FUNCTION_BLOCK FIELDBUS_INT_TO_SIGNAL (* Mirrors IN->OUT if Signal Valid. *)
  (* Standard: 61499-1 *)
  (* Version 1.0, 2026-05-31, franz *)
  PACKAGE logiBUS::signalprocessing::fieldbus;
  IMPORT signalprocessing::FIELDBUS_SIGNAL::NOT_AVAILABLE_WM;
  IMPORT signalprocessing::FIELDBUS_SIGNAL::VALID_SIGNAL_W;
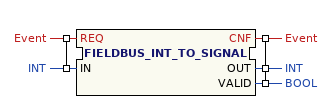
  EVENT_INPUT
    REQ WITH IN; (* Normal Execution Request *)
  END_EVENT
  EVENT_OUTPUT
    CNF WITH OUT, VALID; (* Execution Confirmation *)
  END_EVENT
  VAR_INPUT
    IN : INT := WORD_TO_INT(NOT_AVAILABLE_WM); (* Input *)
  END_VAR
  VAR_OUTPUT
    OUT : INT := 16#0000; (* Output Filtered *)
    VALID : BOOL := FALSE; (* TRUE if Signal is VALID *)
  END_VAR
  EC_STATES
    REQ : REQ -> CNF;
  END_STATES
  ALGORITHM REQ IN ST: (* Executed algorithm *)
IF (IN <= WORD_TO_INT(VALID_SIGNAL_W)) THEN
	OUT := IN;
	VALID := BOOL#TRUE;
ELSE
	OUT := INT#0;
	VALID := BOOL#FALSE;
END_IF;
  END_ALGORITHM
END_FUNCTION_BLOCK
